Staubli VAL3: userPage.dtx

public num nBottomX[2]
  [0] = 17
  [1] = 17
public num nBottomY = 11
num nFirst
num nKey
num nOffSet
num nOldValue[2]
  [0] = 200
  [1] = 200
public num nPage = 10
public num nToSuperV = -1
public num nTopX[2]
  [0] = 21
  [1] = 21
public num nTopY
public num nView
public string sItems = "plo"
string sMessage = "正在保存....请稍等"
public string sTitle = "POLYGON"
public string sToSuperV = "TRAJ m,0"
bool Show
bool bReadWrite = true
public bool bShowDialog
public bool bUseEscape
public bool bUseRefresh
